{attribute 'linkalways'} 
{attribute 'no_explicit_call' := 'This FB is a CLASS and must be accessed using methods or properties'}
{attribute 'enable_dynamic_creation'}
FUNCTION_BLOCK FINAL SUB_LREAL EXTENDS Node
VAR
	in1 : _LREAL(0.0);
	in2 : _LREAL(0.0);
	out : _LREAL(0.0);
END_VAR

METHOD PUBLIC Clone : I_Node
VAR
	pNode : POINTER TO SUB_LREAL;
END_VAR
pNode := __NEW(SUB_LREAL);
Clone := pNode^;
END_METHOD

METHOD FB_init : BOOL
VAR_INPUT
	bInitRetains : BOOL; // if TRUE, the retain variables are initialized (warm start / cold start)
	bInCopyCode : BOOL;  // if TRUE, the instance afterwards gets moved into the copy code (online change)
END_VAR
AddInput('in1',THIS^.in1);
AddInput('in2',THIS^.in2);
AddOutput('out', THIS^.out);
END_METHOD

METHOD PROTECTED OnExecute
VAR
END_VAR
out.Value := in1.Value - in2.Value;
END_METHOD

END_FUNCTION_BLOCK

(* stored: Version 1.1.0.1, ProductVersion 3.1.4024.15
   POU SUB_LREAL: Id {c8bb47a1-7b2f-4038-b8ee-741f0bc3252f}, SpecialFunc None
   Folder Constructor: Id {a5cf67be-9eb7-4c3f-a05f-a7d7ca5ff40c}
   Method Clone: Id {19b0d1df-a76c-4541-9a88-9899ce5a27a8}
   Method FB_init: Id {6321bed3-ca0c-49ca-995d-8a35735dc268}
   Method OnExecute: Id {3649ff5b-d095-4d8b-917d-678b1b1621b9} *)
